TYPE ST_CreateDirBusy :
STRUCT
	isYearBusy : BIT;
	isMonthBusy : BIT;
	isDayBusy : BIT;
	isHourBusy : BIT;
	isMinuteBusy : BIT;
	isSecondBusy : BIT;
END_STRUCT
END_TYPE

(* stored: Version 1.1.0.1, ProductVersion 3.1.4024.12
   DUT ST_CreateDirBusy: Id {41b062ec-3d80-464f-a3aa-b9eecf564718} *)
